TYPE ST_RTDataQRTPacket :
STRUCT
	nSize : UDINT;
	nType : UDINT;
	nTimestamp : LINT;
	nFramenumber : UDINT;
	nComponentCount : UDINT;
END_STRUCT
END_TYPE

(* stored: Version 1.1.0.1, ProductVersion 3.1.4026.8
   DUT ST_RTDataQRTPacket: Id {4535a8f2-5c40-44dd-b06a-d381939bf1e8} *)
